// TIA Portal V17 export
// export: Created 2025-03-05T08:02:57.1965301Z, ExportSetting WithDefaults, DisplayName Totally Integrated Automation Portal, DisplayVersion V17 Update 8, DisplayName TIA Portal Openness, DisplayVersion V17 Update 8, DisplayName TIA Portal Version Control Interface, DisplayVersion V17, DisplayName SINAMICS Startdrive Advanced, DisplayVersion V17 SP2, DisplayName SINAMICS Startdrive G110M, G120, G120C, G120D, G120P, G115D, DisplayVersion V17 SP2, DisplayName SINAMICS Startdrive G130, G150, S120, S150, SINAMICS MV, S210, DisplayVersion V17 SP2, DisplayName STEP 7 Professional, DisplayVersion V17 Update 8, DisplayName SINUMERIK ONE STEP 7 Toolbox, DisplayVersion V17 Update 12, DisplayName SINUMERIK 840D sl STEP 7 Toolbox, DisplayVersion V17 Update 12, DisplayName STEP 7 Safety, DisplayVersion V17 Update 6, DisplayName WinCC Advanced, DisplayVersion V17 Update 8
DATA_BLOCK "DB7300_INTERLOCK"   // DB7300
{ S7_Optimized_Access := 'FALSE'; DB_Accessible_From_OPC_UA := 'FALSE' }
VERSION : 0.1
// stored: AutoNumber false, DBAccessibleFromOPCUA false, DBAccessibleFromWebserver true, IsOnlyStoredInLoadMemory false, IsWriteProtectedInAS false
   VAR
      GENERAL : Struct
         LIFE_BIT : Bool;   // LIFE BIT
         PNEUMATIC_SYSTEM_ON : Bool;   // PNEUMATIC SYSTEM ON
         GAS_SYSTEM_ON : Bool;   // GAS SYSTEM ON
         LASER_UNIT_01_ACTIVE : Bool;   // LASER UNIT 01 ACTIVE
         LASER_UNIT_02_ACTIVE : Bool;   // LASER UNIT 02 ACTIVE
         ASPIRATION_UNIT_01_OK : Bool;   // ASPIRATION UNIT 01 OK
         ASPIRATION_UNIT_02_OK : Bool;   // ASPIRATION UNIT 02 OK
         SELECT_ARGON_GAS : Bool;   // SELECT ARGON GAS
         SELECT_NITROGEN_GAS : Bool;   // SELECT NITROGEN GAS
         SELECT_IMPERIAL_SYSTEM : Bool;   // SELECT IMPERIAL SYSTEM
         SELECT_METRIC_SYSTEM : Bool;   // SELECT METRIC SYSTEM
         CURRENT_PROTECTION_LEVEL : Byte;   // CURRENT ACCESS LEVEL
         EKS_USER : String;   // EKS OPERATOR ID
         EKS_OPERATOR_IDENTIFICATION : Byte;   // EKS OPERATOR IDENTIFICATION
      END_STRUCT;
      POWDER_FEEDERS : Struct
         UNIT_01 : Struct
            U01_PF1_CONDITIONS_OK : Bool;   // UNIT 01 POWDER FEEDER 1 CONDITIONS TO SWITCH ON
            SWITCH_ON_POWDER_UNIT_01 : Bool;   // SWITCH ON POWDER UNIT 01
            SWITCH_OFF_POWDER_UNIT_01 : Bool;   // SWITCH OFF POWDER UNIT 01
            SWITCH_ON_TEMPERATURE_JACKET_UNIT_01 : Bool;   // SWITCH ON TEMPERATURE JACKET UNIT 01
            SWITCH_OFF_TEMPERATURE_JACKET_UNIT_01 : Bool;   // SWITCH OFF TEMPERATURE JACKET UNIT 01
            LASER_MEDICOAT_UNIT_01_ALARM : Bool;   // LASER MEDICOAT UNIT 01 ALARM
            POWDER_FEEDER_1_UNIT_01 : "POWDER FEEDER CNC VALUES SETPOINTS";
         END_STRUCT;
         UNIT_02 : Struct
            U02_PF1_CONDITIONS_OK : Bool;   // UNIT 02 POWDER FEEDER 1 CONDITIONS TO SWITCH ON
            U02_PF2_CONDITIONS_OK : Bool;   // UNIT 02 POWDER FEEDER 2 CONDITIONS TO SWITCH ON
            SWITCH_ON_POWDER_UNIT_02 : Bool;   // SWITCH ON POWDER UNIT 02
            SWITCH_OFF_POWDER_UNIT_02 : Bool;   // SWITCH OFF POWDER UNIT 02
            SWITCH_ON_TEMPERATURE_JACKET_UNIT_02 : Bool;   // SWITCH ON TEMPERATURE JACKET UNIT 02
            SWITCH_OFF_TEMPERATURE_JACKET_UNIT_02 : Bool;   // SWITCH OFF TEMPERATURE JACKET UNIT 02
            LASER_MEDICOAT_UNIT_02_ALARM : Bool;   // LASER MEDICOAT UNIT 02 ALARM
            POWDER_FEEDER_1_UNIT_02 : "POWDER FEEDER CNC VALUES SETPOINTS";
            POWDER_FEEDER_2_UNIT_02 : "POWDER FEEDER CNC VALUES SETPOINTS";
         END_STRUCT;
      END_STRUCT;
      AUX_SIGNALS_INTERFACE : Struct
         LIFE_BIT_FAULT : Bool;   // LIFE BIT COMMUNICATION ALARM
         EMERGENCY_STOPPED : Bool;   // EMERGENCY STOPPED ALARM
         LIFE_SIGN_COUNTER : CTU_INT;   // LIFE SIGN COUNTER
      END_STRUCT;
   END_VAR
BEGIN
END_DATA_BLOCK
